(* CODESYS project Untitled3_RECOVERED_2024-07-11T13-18-48.project

Project tree, tasks and I/O mapping:
  Device : CODESYS Control Win V3, CODESYS, version 3.5.20.10
    application Application
      libraries: Standard, 3.5.18.0 (System)
      task MainTask (cyclic, interval t#20ms, priority 1) calls PLC_PRG
      program PLC_PRG [ST]
*)

// Device/Application/PLC_PRG
PROGRAM PLC_PRG
VAR 
	r_U : REAL;
	r_I : REAL;
	r_S : REAL;
END_VAR

r_S := r_U * r_I;  //Calculate apparent power

END_PROGRAM
